{attribute 'qualified_only'}
VAR_GLOBAL
	fbArbiter: FB_Arbiter(1);
	io_fbFFHWO: FB_HardwareFFOutput;
END_VAR

(* stored: Version 1.1.0.1, ProductVersion 3.1.4022.18
   GVL GVL_PMPS: Id {2a4869fd-2738-48ed-a84f-60d813982319} *)
